ACTION LASTRA_WA_INIT:
Mission^.PPlace	:= cwa; (* valorizzo il punto di deposito *)
(* Aggiorno la struttura delle Lastre in missione *)
Mission^.Slab := WorkAreaState^[Mission^.PPick].Slab[WorkAreaState^[cwa].P];

NLastraDaPrelevare := WorkAreaState^[Mission^.PPick].P-1;
IF NLastraDaPrelevare >= 1 THEN
	NLastraDaPrelevare := 1 ;// añadido para probar
ELSE
	Errore.Code := ErrWA_NumPezzInPrelErrato;
	RETURN;
END_IF


				
Mission^.TPick 	:= TPICK_LASTRA;	// Assegno il tipo di Prelievo
Mission^.XDim 	:= Forming^[WorkAreaState^[Mission^.PPlace].F].PElement[NLastraDaPrelevare].XDim;// WorkAreaState^[Mission^.PPick].Slab[NLastraDaPrelevare].XDim;	// Assegno la dimensione X del pacco presente nel punto di prelievo designato
Mission^.YDim 	:= Forming^[WorkAreaState^[Mission^.PPlace].F].PElement[NLastraDaPrelevare].YDim;//WorkAreaState^[Mission^.PPick].Slab[NLastraDaPrelevare].YDim;	// Assegno la dimensione Y del pacco presente nel punto di prelievo designato
Mission^.ZDim 	:= Forming^[WorkAreaState^[Mission^.PPlace].F].PElement[NLastraDaPrelevare].ZDim;//WorkAreaState^[Mission^.PPick].Slab[NLastraDaPrelevare].ZDim; 	// Assegno la dimensione Z del pacco presente nel punto di prelievo designato
ppick := Mission^.PPick;

IF Mission^.XDim <=0	OR Mission^.YDim <= 0 THEN
	Errore.Code := ErrEsMisionSinDimesionPieza;
	RETURN;
END_IF
(* Valorizzazione del lato di prelievo nel caso di prelievo su cavallina *)
IF WorkareaState^[Mission^.PPick].Supporto.Tipologia = e_Tipo_Pallet.BUNDLE THEN //Se ho in prelievo il supporto di tipo bundle
	IF ppickOld <> Mission^.PPick THEN 	//Ad ogni cambio di postazione setto il valore del lato iniziale a 0
		TFClearApprendimento(ADR(WorkAreaState^[Mission^.PPick].Apprendimento));//Pulisco la struttura dell'apprendimento
		LatoPrelievo := 180;				//Vado a prelevare sul lato 180	
		TFWAM_CreaMissione_PrelLastraDaWA.Quota_FormaturaJ := 180; //Assegno la quota di 0° per il prelievo, in questo modo la pinza parte a fare il tasteggio in questa posizione					
		IF LatoPrelievo = 0 THEN
		(* Apprendimento lungo X *)
			WorkAreaState^[Mission^.PPick].Apprendimento.X.Lato0.Stato		:= APPRENDIMENTO_DISABILITATO;
			WorkAreaState^[Mission^.PPick].Apprendimento.Y.Lato0.Stato		:= APPRENDIMENTO_DA_ESEGUIRE;
		ELSIF LatoPrelievo = 180 THEN
			WorkAreaState^[Mission^.PPick].Apprendimento.X.Lato180.Stato	:= APPRENDIMENTO_DISABILITATO;
			WorkAreaState^[Mission^.PPick].Apprendimento.Y.Lato180.Stato	:= APPRENDIMENTO_DA_ESEGUIRE;
		END_IF
	ELSE
		LatoPrelievo := 180;				//Vado a prelevare sul lato 180	
		TFWAM_CreaMissione_PrelLastraDaWA.Quota_FormaturaJ := 180; //Assegno la quota di 0° per il prelievo, in questo modo la pinza parte a fare il tasteggio in questa posizione					
		IF LatoPrelievo = 0 THEN
		(* Apprendimento lungo X *)
			WorkAreaState^[Mission^.PPick].Apprendimento.X.Lato0.Stato		:= APPRENDIMENTO_DISABILITATO;
			IF WorkAreaState^[Mission^.PPick].Apprendimento.Y.Lato0.Stato <> APPRENDIMENTO_ESEGUITO THEN
				WorkAreaState^[Mission^.PPick].Apprendimento.Y.Lato0.Stato		:= APPRENDIMENTO_DA_ESEGUIRE;
			END_IF
		ELSIF LatoPrelievo = 180 THEN
			WorkAreaState^[Mission^.PPick].Apprendimento.X.Lato180.Stato	:= APPRENDIMENTO_DISABILITATO;
			IF WorkAreaState^[Mission^.PPick].Apprendimento.Y.Lato180.Stato <> APPRENDIMENTO_ESEGUITO THEN
				WorkAreaState^[Mission^.PPick].Apprendimento.Y.Lato180.Stato	:= APPRENDIMENTO_DA_ESEGUIRE;
			END_IF
		END_IF
	END_IF
ELSIF WorkareaState^[Mission^.PPick].Supporto.Tipologia = e_Tipo_Pallet.CAVALLETTO THEN //Se ho in prelievo il supporto di tipo cavalletto
	
	AguloDeRecogida := FunLadoTrabajoCaballete(Piezas_LadoA := 
						HMI_NumeroPezziPresentiCavallete[Mission^.PPick].HMI_NumeroPezziPresentiPostazione_A_Cavaleto , 
								Piezas_Ladob := HMI_NumeroPezziPresentiCavallete[Mission^.PPick].HMI_NumeroPezziPresentiPostazione_B_Cavaleto ,
								Recoger := TRUE ,dejar := FALSE ,GestionLadoTrabajo := WorkareaState^[Mission^.PPick].Supporto.TipoTrabajoLado_Cavallete);
	LatoPrelievo := AguloDeRecogida ;
	IF FALSE THEN 
			IF FormaturaAFRAMERT[WorkAreaState^[Mission^.PPlace].F].PElement[WorkAreaState^[Mission^.PPick].P-1].J > 90 THEN
				LatoPrelievo := 180;
			
			ELSIF FormaturaAFRAMERT[WorkAreaState^[Mission^.PPlace].F].PElement[WorkAreaState^[Mission^.PPick].P-1].J  < 90 THEN
				LatoPrelievo := 0;
			END_IF	
	END_IF
	
	IF ppickOld <> Mission^.PPick THEN 	//Ad ogni cambio di postazione setto il valore del lato iniziale a 0
		TFClearApprendimento(ADR(WorkAreaState^[Mission^.PPick].Apprendimento));//Pulisco la struttura dell'apprendimento
		TFWAM_CreaMissione_PrelLastraDaWA.Quota_FormaturaJ := 180; //Assegno la quota di 0° per il prelievo, in questo modo la pinza parte a fare il tasteggio in questa posizione					
		WorkAreaState^[Mission^.PPick].Apprendimento.X.Lato0.Stato		:= APPRENDIMENTO_DISABILITATO;
		WorkAreaState^[Mission^.PPick].Apprendimento.Y.Lato0.Stato		:= APPRENDIMENTO_DA_ESEGUIRE;
		WorkAreaState^[Mission^.PPick].Apprendimento.X.Lato180.Stato	:= APPRENDIMENTO_DISABILITATO;
		WorkAreaState^[Mission^.PPick].Apprendimento.Y.Lato180.Stato	:= APPRENDIMENTO_DA_ESEGUIRE;
	ELSE
		TFWAM_CreaMissione_PrelLastraDaWA.Quota_FormaturaJ := 180; //Assegno la quota di 0° per il prelievo, in questo modo la pinza parte a fare il tasteggio in questa posizione					
		IF LatoPrelievo = 0 THEN
		(* Apprendimento lungo X *)
			WorkAreaState^[Mission^.PPick].Apprendimento.X.Lato0.Stato		:= APPRENDIMENTO_DISABILITATO;
			IF WorkAreaState^[Mission^.PPick].Apprendimento.Y.Lato0.Stato <> APPRENDIMENTO_ESEGUITO THEN
				WorkAreaState^[Mission^.PPick].Apprendimento.Y.Lato0.Stato		:= APPRENDIMENTO_DA_ESEGUIRE;
				//WorkAreaState^[Mission^.PPick].Apprendimento.Y.Lato0.QuotaStart	:= 1000;
			END_IF
		ELSIF LatoPrelievo = 180 THEN
			WorkAreaState^[Mission^.PPick].Apprendimento.X.Lato180.Stato	:= APPRENDIMENTO_DISABILITATO;
			IF WorkAreaState^[Mission^.PPick].Apprendimento.Y.Lato180.Stato <> APPRENDIMENTO_ESEGUITO THEN
				WorkAreaState^[Mission^.PPick].Apprendimento.Y.Lato180.Stato	:= APPRENDIMENTO_DA_ESEGUIRE;
				//WorkAreaState^[Mission^.PPick].Apprendimento.Y.Lato180.QuotaStart	:= 1000;
			END_IF
		END_IF
	END_IF
ELSIF WorkareaState^[Mission^.PPick].Supporto.Tipologia <> e_Tipo_Pallet.CAVALLETTO AND WorkareaState^[Mission^.PPick].Supporto.Tipologia <> e_Tipo_Pallet.BUNDLE THEN //Se NON ho in prelievo il supporto di tipo cavalletto
	LatoPrelievo := 90; //Setto il lato di prelievo = 90
	IF ppickOld <> ppick THEN 	//Ad ogni cambio di postazione setto il valore del lato iniziale a 0
		TFClearApprendimento(ADR(WorkAreaState^[Mission^.PPick].Apprendimento));//Pulisco la struttura dell'apprendimento
	END_IF
	TFWAM_CreaMissione_PrelLastraDaWA.Quota_FormaturaJ := 90;//Assegno la quota di 90° per il prelievo, in questo modo la pinza preleverà in orizzontale
	IF WorkAreaState^[Mission^.PPick].Apprendimento.Z.Lato90.Stato <> APPRENDIMENTO_ESEGUITO THEN
		WorkAreaState^[Mission^.PPick].Apprendimento.Z.Lato90.Stato := APPRENDIMENTO_DA_ESEGUIRE;
		IF WorkareaState^[Mission^.PPick].Supporto.Tipologia = e_Tipo_Pallet.CASSA_STANDARD THEN 
			WorkAreaState^[Mission^.PPick].Apprendimento.Z.Lato90.QuotaStart 	:= 700;
		ELSE
			WorkAreaState^[Mission^.PPick].Apprendimento.Z.Lato90.QuotaStart 	:= 700;
		END_IF
	END_IF
END_IF

//Disabilito apprendimento in deposito se disabilitato
IF NOT HMI_AbilitaDepositoPaccoOrrizzontaleConTasteggio AND FALSE THEN
	WorkAreaState^[Mission^.PPick].Apprendimento.Z.Lato90.Stato := APPRENDIMENTO_DISABILITATO;	
END_IF

(* Memorizzo l'ultima postazione in cui è stato effettuato il prelievo *)
UltimaPostazioneInPrelievo := Mission^.PPick;
ppickOld := Mission^.PPick;

//Z prelievo a seconda della tipologia 
IF WorkareaState^[Mission^.PPick].Supporto.Tipologia = e_Tipo_Pallet.BUNDLE THEN //SE PRELIEVO SU BUNDLE O CASSA
	IF LatoPrelievo = 180 THEN
		AngoloPrelievo 					:= 180-2;
		AltezzaCentroLastraInclinata 	:=  	ABS((Mission^.YDim/2) * COS(DEG_TO_RAD(AngoloPrelievo)));
		QuotaLastraYRealTimePrelievo 			:= FormaturaBundleRT[WorkAreaProductionList^[Mission^.PPlace].NumeroListaAssociata].PElement[WorkAreaState^[Mission^.PPick].P-1].Y;
		QuotaLastraZRealTimePrelievo 			:= FormaturaBundleRT[WorkAreaProductionList^[Mission^.PPlace].NumeroListaAssociata].PElement[WorkAreaState^[Mission^.PPick].P-1].Z (*+  (*Dimensioni_Pinza.DimTraveVerticale / 2*) CuotaOffSetZRecogidaBundel *);
	ELSIF LatoPrelievo = 0 THEN
		AngoloPrelievo 							:= 2;
		AltezzaCentroLastraInclinata 			:=  ABS((Mission^.YDim/2) * COS(DEG_TO_RAD(AngoloPrelievo)));
		IF TRUE THEN 
			QuotaLastraYRealTimePrelievo 			:= FormaturaBundleRT[WorkAreaProductionList^[Mission^.PPlace].NumeroListaAssociata].PElement[WorkAreaState^[Mission^.PPick].P_Cava.HMI_NumeroPezziPresentiPostazione_A_Cavaleto-1].CooCavallete.LadoA.CoordenadaFinale_Y;
			QuotaLastraZRealTimePrelievo 			:= FormaturaBundleRT[WorkAreaProductionList^[Mission^.PPlace].NumeroListaAssociata].PElement[WorkAreaState^[Mission^.PPick].P_Cava.HMI_NumeroPezziPresentiPostazione_A_Cavaleto-1].CooCavallete.LadoA.CoordenadaFinale_Z;(*+  (*Dimensioni_Pinza.DimTraveVerticale / 2*) CuotaOffSetZRecogidaBundel *);
		ELSE
			QuotaLastraYRealTimePrelievo 			:= FormaturaBundleRT[WorkAreaProductionList^[Mission^.PPlace].NumeroListaAssociata].PElement[WorkAreaState^[Mission^.PPick].P-1].Y;
			QuotaLastraZRealTimePrelievo 			:= FormaturaBundleRT[WorkAreaProductionList^[Mission^.PPlace].NumeroListaAssociata].PElement[WorkAreaState^[Mission^.PPick].P-1].Z (*+ (*Dimensioni_Pinza.DimTraveVerticale / 2*) CuotaOffSetZRecogidaBundel*) ;		
			
		END_IF
		
	ELSE
		AngoloPrelievo := 90;
		AltezzaCentroLastraInclinata := 0;
		QuotaLastraZRealTimePrelievo := 0;
		QuotaLastraYRealTimePrelievo := 0;
	END_IF
ELSIF WorkareaState^[Mission^.PPick].Supporto.Tipologia = e_Tipo_Pallet.CAVALLETTO THEN
	IF LatoPrelievo = 180 THEN
		AngoloPrelievo 					:= 180-2;
		AltezzaCentroLastraInclinata 	:= ABS((Mission^.YDim/2) * COS(DEG_TO_RAD(AngoloPrelievo)));
		IF TRUE THEN
			QuotaLastraYRealTimePrelievo 			:= FormaturaAFRAMERT[WorkAreaProductionList^[Mission^.PPlace].NumeroListaAssociata].PElement[WorkAreaState^[Mission^.PPick].P_Cava.HMI_NumeroPezziPresentiPostazione_B_Cavaleto-1].CooCavallete.LadoB.CoordenadaFinale_Y;
			QuotaLastraZRealTimePrelievo 			:= FormaturaAFRAMERT[WorkAreaProductionList^[Mission^.PPlace].NumeroListaAssociata].PElement[WorkAreaState^[Mission^.PPick].P_Cava.HMI_NumeroPezziPresentiPostazione_B_Cavaleto-1].CooCavallete.LadoB.CoordenadaFinale_Z;(*+  (*Dimensioni_Pinza.DimTraveVerticale / 2*) CuotaOffSetZRecogidaBundel *);
		ELSE
 			QuotaLastraYRealTimePrelievo 			:= FormaturaAFRAMERT[WorkAreaProductionList^[Mission^.PPlace].NumeroListaAssociata].PElement[WorkAreaState^[Mission^.PPick].P-1].Y;
			QuotaLastraZRealTimePrelievo 			:= FormaturaAFRAMERT[WorkAreaProductionList^[Mission^.PPlace].NumeroListaAssociata].PElement[WorkAreaState^[Mission^.PPick].P-1].Z + (*Dimensioni_Pinza.DimTraveVerticale / 2*) CuotaOffSetZRecogidaCaballete;
		END_IF
	ELSIF LatoPrelievo = 0 THEN
		AngoloPrelievo 					:= 3;
		AltezzaCentroLastraInclinata 	:= ABS((Mission^.YDim/2) * COS(DEG_TO_RAD(AngoloPrelievo)));
		IF TRUE THEN 
			QuotaLastraYRealTimePrelievo 			:= FormaturaAFRAMERT[WorkAreaProductionList^[Mission^.PPlace].NumeroListaAssociata].PElement[WorkAreaState^[Mission^.PPick].P_Cava.HMI_NumeroPezziPresentiPostazione_A_Cavaleto-1].CooCavallete.LadoA.CoordenadaFinale_Y;
			QuotaLastraZRealTimePrelievo 			:= FormaturaAFRAMERT[WorkAreaProductionList^[Mission^.PPlace].NumeroListaAssociata].PElement[WorkAreaState^[Mission^.PPick].P_Cava.HMI_NumeroPezziPresentiPostazione_A_Cavaleto-1].CooCavallete.LadoA.CoordenadaFinale_Z;(*+  (*Dimensioni_Pinza.DimTraveVerticale / 2*) CuotaOffSetZRecogidaBundel *);
		ELSE
			QuotaLastraYRealTimePrelievo 			:= FormaturaAFRAMERT[WorkAreaProductionList^[Mission^.PPlace].NumeroListaAssociata].PElement[WorkAreaState^[Mission^.PPick].P-1].Y;
			QuotaLastraZRealTimePrelievo 			:= FormaturaAFRAMERT[WorkAreaProductionList^[Mission^.PPlace].NumeroListaAssociata].PElement[WorkAreaState^[Mission^.PPick].P-1].Z (*+ (*Dimensioni_Pinza.DimTraveVerticale / 2*) CuotaOffSetZRecogidaCaballete *);
		END_IF
	ELSE
		AngoloPrelievo := 90;
		AltezzaCentroLastraInclinata := 0;
		QuotaLastraZRealTimePrelievo := 0;
		QuotaLastraYRealTimePrelievo := 0;
	END_IF
ELSE
	IF LatoPrelievo = 90 THEN		
		AngoloPrelievo := 90;
		AltezzaCentroLastraInclinata := 0;
		QuotaLastraZRealTimePrelievo := 0;
		QuotaLastraYRealTimePrelievo := 0;
	ELSE
		Errore.Code := ErrWA_SupportoInPrelivoNonPrevisto;
	END_IF
END_IF

//CALCOLO INGOMBRI PINZA						

;
//OffSetZRecogidaEnAngulo				:=  -20 ;					
//ScostamentoVerticalePuntoCentrale := ABS(Dimensioni_Pinza.Spessore * COS(deg_to_rad(-90+AngoloPrelievo))-Dimensioni_Pinza.Spessore);

// Calculo Del Ingombro Pinza Mision Recogida lastra
TFCalcoliIngombroPinza(Mission := Mission,
						WorkAreaManager := WorkAreaManager,
						WorkAreaState := ADR(WorkAreaState),
						ModuleAX_J := ModuleAX_J,
						AngoloRotazioneDestinazionePinza:= LatoPrelievo,//Forming^[WorkAreaState^[Mission^.PPlace].F].PElement[WorkAreaState^[Mission^.PPlace].P].J+2,
						IngombroX_Pos 				:= ADR(IngombroX_Pos),
						IngombroY_Pos 				:= ADR(IngombroY_Pos),
						IngombroX_Neg 				:= ADR(IngombroX_Neg),
						IngombroY_Neg 				:= ADR(IngombroY_Neg),
						IngombroZ_Pos 				:= ADR(IngombroZ_Pos),
						IngombroZ_Neg 				:= ADR(IngombroZ_Neg),
						IngombroY_Tot 				:= ADR(IngombroY_Tot),
						IngombroDestinazioneX_Pos 	:= ADR(IngombroDestinazioneX_Pos),
						IngombroDestinazioneY_Pos 	:= ADR(IngombroDestinazioneY_Pos),
						IngombroDestinazioneX_Neg 	:= ADR(IngombroDestinazioneX_Neg),
						IngombroDestinazioneY_Neg 	:= ADR(IngombroDestinazioneY_Neg),
						IngombroDestinazioneZ_Pos 	:= ADR(IngombroDestinazioneZ_Pos),
						IngombroDestinazioneZ_Neg 	:= ADR(IngombroDestinazioneZ_Neg),
						IngombroMaxX_Pos 			:= ADR(IngombroMaxX_Pos),
						IngombroMaxY_Pos 			:= ADR(IngombroMaxY_Pos),
						IngombroMaxX_Neg 			:= ADR(IngombroMaxX_Neg),
						IngombroMaxY_Neg 			:= ADR(IngombroMaxY_Neg),
						IngombroMaxZ_Pos 			:= ADR(IngombroMaxZ_Pos),
						IngombroMaxZ_Neg 			:= ADR(IngombroMaxZ_Neg),
						IngombroY_Pos_0  			:= ADR(IngombroY_Pos_0),		 		
						IngombroY_Neg_180 			:= ADR(IngombroY_Neg_180),
						IngombroY_Neg_0 			:= ADR(IngombroY_Neg_0),	
						IngombroY_Pos_180 			:= ADR(IngombroY_Pos_180),
						ScostamentoVerticalePuntoCentrale := ADR(ScostamentoVerticalePuntoCentrale));





(* Assegnazione quote alla Missione *)
TFWAM_CreaMissione_PrelLastraDaWA(NPosInLavoro				:= Mission^.PPick, //Numero Postazione di lavoro
									Angolo_Destinazione 	:= LatoPrelievo, //Angolo di deposito dell'elemento
									PosizioneAttuale_X      := ModuleAX_X^.Ax^.Status.ActPosition, //Posizione attuale asse X
									TipologiaTraiettoria    := TRAIETTORIA_CON_APPROCCIO,//Forming^[WorkAreaState^[cwa].F].PElement[WorkAreaState^[cwa].P].Trajectory,
									Apprendimento			:= WorkAreaState^[Mission^.PPick].Apprendimento,
									CicloDiPrelievo         := TRUE,
									HmaxElemento			:= WorkAreaState^[Mission^.PPick].Supporto.HMAX,
									Offset_Apprendimento_X 	:= 0,//OffsetApprendimento.Lastra.X, //Offset X Postazione,
									Offset_Apprendimento_Y 	:= OffsetApprendimento.Lastra.Y, //Offset Y Postazione
									Offset_Apprendimento_Z 	:= OffsetApprendimento.Lastra.Z, //Offset Z Postazione
									Offset_Apprendimento_J 	:= 0,//OffsetApprendimento.Lastra.J, //Offset J Postazione

									Quota_PostX				:= WorkArea^[Mission^.PPick].X, //Quota X Postazione
									Quota_PostY				:= WorkArea^[Mission^.PPick].Y, //Quota Y Postazione
									Quota_PostZ				:= WorkArea^[Mission^.PPick].Z, //Quota Z Postazione
									Quota_PostJ				:= WorkArea^[Mission^.PPick].Rx, //Quota J Postazione
									
									Offset_Postazione_X 	:= WorkAreaOffset^[Mission^.PPick].X, //Offset X Postazione
									Offset_Postazione_Y 	:= WorkAreaOffset^[Mission^.PPick].Y, //Offset Y Postazione
									Offset_Postazione_Z 	:= WorkAreaOffset^[Mission^.PPick].Z, //Offset Z Postazione
									Offset_Postazione_J 	:= WorkAreaOffset^[Mission^.PPick].Rx, //Offset J Postazione
									
									Pallet_DimX				:= WorkAreaState^[Mission^.PPick].Supporto.XDim, //Dimensione X Pallet
									Pallet_DimY				:= WorkAreaState^[Mission^.PPick].Supporto.YDim, //Dimensione Y Pallet
									Pallet_DimZ				:= WorkAreaState^[Mission^.PPick].Supporto.ZDim, //Dimensione Z Pallet
									Pallet_DimBaseUtile		:= WorkAreaState^[Mission^.PPick].Supporto.DimBaseUtile, //Dimensione Z Pallet
									
									Offset_Pallet_X_0		:= 0,//Forming^[WorkAreaState^[Mission^.PPlace].F].Pallet.OFSDE_X0, //Offset X Pallet o Casse
									Offset_Pallet_Y_0		:= 0,//Forming^[WorkAreaState^[Mission^.PPlace].F].Pallet.OFSDE_Y0, //Offset Y Pallet o Casse 
									Offset_Pallet_Z_0		:= OffSetZRecogidaEnAngulo0,//Forming^[WorkAreaState^[Mission^.PPlace].F].Pallet.OFSDE_Z0, //Offset Z Pallet o Casse + è grande + il deposito si distanzia dal supporto
									Offset_Pallet_J_0		:= 0,//Forming^[WorkAreaState^[Mission^.PPlace].F].Pallet.OFSDE_J0, //Offset J Pallet o Casse + è grande + la lastra sarà inclinata verso l'angolo crescente
															   
									Offset_Pallet_X_90		:= 0,//Forming^[WorkAreaState^[Mission^.PPlace].F].Pallet.OFSDE_X90, //Offset X Pallet lato 0-90 
									Offset_Pallet_Y_90		:= 0,//Forming^[WorkAreaState^[Mission^.PPlace].F].Pallet.OFSDE_Y90, //Offset Y Pallet lato 0-90 + è grande + il deposito si distanzia dal supporto
									Offset_Pallet_Z_90		:= 0,//Forming^[WorkAreaState^[Mission^.PPlace].F].Pallet.OFSDE_Z90, //Offset Z Pallet lato 0-90 + è grande + il deposito si distanzia dal supporto
									Offset_Pallet_J_90		:= 0,//Forming^[WorkAreaState^[Mission^.PPlace].F].Pallet.OFSDE_J90, //Offset J Pallet lato 0-90 + è grande + la lastra sarà inclinata in fase di deposito
															  
									Offset_Pallet_X_180		:= 0,//Forming^[WorkAreaState^[Mission^.PPlace].F].Pallet.OFSDE_X180, //Offset X Pallet lato 90-180
									Offset_Pallet_Y_180		:= 0,//Forming^[WorkAreaState^[Mission^.PPlace].F].Pallet.OFSDE_Y180, //Offset Y Pallet lato 90-180 + è grande + il deposito si distanzia dal supporto
									Offset_Pallet_Z_180		:= OffSetZRecogidaEnAngulo180,//Forming^[WorkAreaState^[Mission^.PPlace].F].Pallet.OFSDE_Z180, //Offset Z Pallet lato 90-180 + è grande + il deposito si distanzia dal supporto
									Offset_Pallet_J_180		:= 0,//Forming^[WorkAreaState^[Mission^.PPlace].F].Pallet.OFSDE_J180, //Offset J Pallet lato 90-180 + è grande + la lastra sarà inclinata in fase di deposito
									
									Quota_FormaturaX 		:= 0,//Quota  X da Formatura
									Quota_FormaturaY 		:= ABS(QuotaLastraYRealTimePrelievo),//Quota  Y da Formatura
									Quota_FormaturaZ 		:= QuotaLastraZRealTimePrelievo,//Quota  Z da Formatura
									Quota_FormaturaJ 		:= LatoPrelievo,//Quota  Z da Formatura
									
									Distanza_ApproccioFormaturaX 		:= PickPlaceParameters^.XPickApproach,
									Distanza_ApproccioFormaturaY 		:= PickPlaceParameters^.YPickApproach, 
									Distanza_ApproccioFormaturaZ 		:= PickPlaceParameters^.ZPickApproach,
									Distanza_ApproccioFormaturaJ 		:= PickPlaceParameters^.JPickApproach,
									
									Quota_DestX 			=> Mission^.XPick, //Quota DESTINAZIONE X
									Quota_DestY 			=> Mission^.YPick, //Quota DESTINAZIONE Y
									Quota_DestZ 			=> Mission^.ZPick, //Quota DESTINAZIONE Z
									Quota_DestJ 			=> Mission^.JPick, //Quota DESTINAZIONE J	
									
									Quota_ApproccioDestX 	=> Mission^.XPickApproach, //Quota APPROCCIO di DESTINAZIONE X
									Quota_ApproccioDestY 	=> Mission^.YPickApproach, //Quota APPROCCIO di DESTINAZIONE Y
									Quota_ApproccioDestZ 	=> Mission^.ZPickApproach, //Quota APPROCCIO di DESTINAZIONE Z
									Quota_ApproccioDestJ 	=> Mission^.JPickApproach);//Quota APPROCCIO di DESTINAZIONE J	

//Valorizziamo il preleivo di z a una quota positiva per evitare errori di interferenza									
IF LatoPrelievo = 90 THEN
	IF Mission^.ZPick <= 0 THEN
		Mission^.ZPick := ModuleAX_Z^.AxisPar^.MinPosition;
	END_IF
END_IF 		
//
IF LatoPrelievo = 180 THEN
	
	IF HMI_OffsetDepositoLastra.J180 = 0 OR  HMI_OffsetDepositoLastra.J180 < 0 THEN 
		Mission^.JPick := 180 - 2;
	ELSIF HMI_OffsetDepositoLastra.J180 <= 4 AND   HMI_OffsetDepositoLastra.J180 > 0 THEN 
		Mission^.JPick := 180 - HMI_OffsetDepositoLastra.J180;
	ELSE 
		Mission^.JPick := 180 - 2;	
	END_IF
	


	
	
	
	//IF WorkAreaState^[Mission^.PPick].Apprendimento.Y.Lato180.Stato = APPRENDIMENTO_ESEGUITO THEN
	//	Mission^.YPickApproach	:= MIN(Mission^.YPickApproach,WorkAreaState^[Mission^.PPick].Supporto.YDim + IngombroDestinazioneY_Neg);
	//ELSE
	//	Mission^.YPickApproach	:= WorkArea^[Mission^.PPick].Y + WorkAreaState^[Mission^.PPick].Supporto.YDim + IngombroDestinazioneY_Neg - 50;
	//end_if
	//&&&&&&&&&&&&&&&&&&&&&&&&&&&&&&&&&&&&&&&&&&&&&&&&&&&&&&&&&&&&&&&&&&&&&&&&&&&&&
	//Mission^.YPick 				:= Mission^.YPick - 80 ;	// modificado = 200
	//&&&&&&&&&&&&&&&&&&&&&&&&&&&&&&&&&&&&&&&&&&&&&&&&&&&&&&&&&&&&&&&&&&&&&&&&&&&&&&&&&&&&
	IF WorkareaState^[Mission^.PPick].Supporto.Tipologia = e_Tipo_Pallet.BUNDLE THEN //SE PRELIEVO SU BUNDLE O CASSA
		Y_PuntoPrelievo180 := Mission^.YPick ;
			Z_PuntoPrelievo180Bundle    := Mission^.ZPick ;
		 IF Mission^.YDim  < 1300 THEN
			Mission^.YPick 				:= Mission^.YPick - (80  ) ; //(Dimensioni_Pinza.DimTraveVerticale /2) (*-80*);	// modificado = 200
			Mission^.ZPick				:= Mission^.ZPick + (15 +25) ;
			Mission^.ZPickApproach		:= Mission^.ZPick;
			ELSE
				
			Mission^.YPick 				:= Mission^.YPick  - (45) ; //(Dimensioni_Pinza.DimTraveVerticale /2) (*-80*);	// modificado = 200
 			Mission^.ZPick				:= Mission^.ZPick + 15 ;
			Mission^.ZPickApproach		:= Mission^.ZPick;
		 END_IF
		
	
		
	ELSIF WorkareaState^[Mission^.PPick].Supporto.Tipologia = e_Tipo_Pallet.CAVALLETTO THEN //Se ho in prelievo il supporto di tipo cavalletto	
		Y_PuntoPrelievo180 := Mission^.YPick ;
		Z_PuntoPrelievo180Bundle    := Mission^.ZPick ;
		IF Mission^.YDim  < 1300 THEN
				Mission^.YPick 				:= Mission^.YPick - (Dimensioni_Pinza.DimTraveVerticale -35) ;//(Dimensioni_Pinza.DimTraveVerticale /2) (*-70*)  ;	// modificado = 200
				Mission^.ZPick				:= Mission^.ZPick + (25 +20) ;
				Mission^.ZPickApproach		:= Mission^.ZPick;		
			ELSE
				Mission^.YPick 				:= Mission^.YPick - 60 ; //(Dimensioni_Pinza.DimTraveVerticale /2) (*-70*)  ;	// modificado = 200
				Mission^.ZPick				:= Mission^.ZPick + 28 ;
				Mission^.ZPickApproach		:= Mission^.ZPick;		
			
		END_IF
		
		
	END_IF

ELSIF LatoPrelievo = 0 THEN
	//Mission^.JPick := 3;
	IF HMI_OffsetDepositoLastra.J0 > 4 THEN 
		Mission^.JPick := 4;
	ELSIF HMI_OffsetDepositoLastra.J0 <> 0 THEN 
		Mission^.JPick := HMI_OffsetDepositoLastra.J0;	
	ELSIF HMI_OffsetDepositoLastra.J0 = 0 THEN 
		Mission^.JPick := 3;	
	END_IF
	Y_PuntoPrelievo0 := Mission^.YPick ;
	
	Z_PuntoPrelievo180Bundle    := Mission^.ZPick ;
	IF Mission^.YDim  < 1300 THEN
			Mission^.YPick 				:= Mission^.YPick -0 ; // + 50 (*+ 50 *);
			Mission^.ZPick				:= Mission^.ZPick + (20) ; // pieza pequeña
			Mission^.ZPickApproach		:= Mission^.ZPick;
		ELSE
			Mission^.YPick 				:= Mission^.YPick  + 25; // + 50 (*+ 50 *);
			Mission^.ZPick				:= Mission^.ZPick + 12 ;
			Mission^.ZPickApproach		:= Mission^.ZPick;	
	END_IF
	
	
	
END_IF											 			
//									
IF TFWAM_CreaMissione_PrelLastraDaWA.Errore.Code > 0 THEN
	Errore := TFWAM_CreaMissione_PrelLastraDaWA.Errore;
	WorkAreaManager^.State 	:= WAMANAGER_NOP;	// setto lo stato del WAMANAGER
	RETURN;//EXIT;
END_IF	

(* Valorizzazione del lato di prelievo nel caso di depostio su cavallina *)
IF WorkareaState^[Mission^.PPlace].Supporto.Tipologia = e_Tipo_Pallet.CAVALLETTO THEN //Se ho in prelievo il supporto di tipo cavalletto
	
	AguloDeDeposito := FunLadoTrabajoCaballete(Piezas_LadoA := 
						HMI_NumeroPezziPresentiCavallete[Mission^.PPlace].HMI_NumeroPezziPresentiPostazione_A_Cavaleto , 
								Piezas_Ladob := HMI_NumeroPezziPresentiCavallete[Mission^.PPlace].HMI_NumeroPezziPresentiPostazione_B_Cavaleto ,
								Recoger := FALSE ,dejar := TRUE, GestionLadoTrabajo := WorkareaState^[Mission^.PPlace].Supporto.TipoTrabajoLado_Cavallete);
	LatoDeposito := AguloDeDeposito ;

	IF FALSE THEN
		IF FormaturaAFRAMERT[WorkAreaState^[Mission^.PPlace].F].PElement[WorkAreaState^[Mission^.PPlace].P].J > 90 THEN
			LatoDeposito := 180;
		
		ELSIF FormaturaAFRAMERT[WorkAreaState^[Mission^.PPlace].F].PElement[WorkAreaState^[Mission^.PPlace].P].J  < 90 THEN
			LatoDeposito := 0;
		END_IF
	END_IF
	
	
ELSIF WorkareaState^[Mission^.PPlace].Supporto.Tipologia = e_Tipo_Pallet.BUNDLE THEN
	LatoDeposito := 180;
ELSIF WorkareaState^[Mission^.PPlace].Supporto.Tipologia <> e_Tipo_Pallet.CAVALLETTO AND WorkareaState^[Mission^.PPlace].Supporto.Tipologia <> e_Tipo_Pallet.BUNDLE THEN //Se NON ho in prelievo il supporto di tipo cavalletto
	IF PplaceOld <> Mission^.PPlace THEN 	//Ad ogni cambio di postazione setto il valore del lato iniziale a 0
		TFClearApprendimento(ADR(WorkAreaState^[Mission^.PPlace].Apprendimento));//Pulisco la struttura dell'apprendimento
	END_IF
	LatoDeposito := 90; //Setto il lato di prelievo = 90
	TFWAM_CreaMissione_PrelLastraDaWA.Quota_FormaturaJ := 90;//Assegno la quota di 90° per il prelievo, in questo modo la pinza preleverà in orizzontale
	IF WorkAreaState^[Mission^.PPlace].Apprendimento.Z.Lato90.Stato <> APPRENDIMENTO_ESEGUITO THEN
		WorkAreaState^[Mission^.PPlace].Apprendimento.Z.Lato90.Stato := APPRENDIMENTO_DA_ESEGUIRE;
		IF WorkareaState^[Mission^.PPlace].Supporto.Tipologia = e_Tipo_Pallet.CASSA_STANDARD THEN 
			WorkAreaState^[Mission^.PPlace].Apprendimento.Z.Lato90.QuotaStart 	:= 700;
		ELSE
			WorkAreaState^[Mission^.PPlace].Apprendimento.Z.Lato90.QuotaStart 	:= 700;
		END_IF
	END_IF
END_IF

//Disabilito apprendimento in deposito se disabilitato
IF NOT HMI_AbilitaDepositoPaccoOrrizzontaleConTasteggio AND FALSE THEN
	WorkAreaState^[Mission^.PPlace].Apprendimento.Z.Lato90.Stato := APPRENDIMENTO_DISABILITATO;	
END_IF

//mettiamo un offset sul deposito bundle
IF LatoDeposito = 180 THEN
	TFWAM_CreaMissione_DepLastraDaWA.Offset_Pallet_Y_0 := 0;// HMI_OffsetDepositoLastra.Y0;
	TFWAM_CreaMissione_DepLastraDaWA.Offset_Pallet_Z_0 := 0;//HMI_OffsetDepositoLastra.Z0;
	TFWAM_CreaMissione_DepLastraDaWA.Offset_Pallet_Y_0 := 0;

	TFWAM_CreaMissione_DepLastraDaWA.Offset_Pallet_Y_180 := HMI_OffsetDepositoLastra.Y180;
	TFWAM_CreaMissione_DepLastraDaWA.Offset_Pallet_Z_180 := HMI_OffsetDepositoLastra.Z180;
	TFWAM_CreaMissione_DepLastraDaWA.Offset_Pallet_Z_90  := 0;
	AngoloDepositoLastra := 180; // := 180-1; Modificado 16-6-2025
ELSIF LatoDeposito = 90 THEN
	TFWAM_CreaMissione_DepLastraDaWA.Offset_Pallet_Y_180 := 0;
	TFWAM_CreaMissione_DepLastraDaWA.Offset_Pallet_Z_180 := 0;
	TFWAM_CreaMissione_DepLastraDaWA.Offset_Pallet_Y_180 := 0;
	IF NOT HMI_AbilitaDepositoPaccoOrrizzontaleConTasteggio THEN
		TFWAM_CreaMissione_DepLastraDaWA.Offset_Pallet_Z_90  := (* 30 +*) HMI_OffsetDepositoLastra.Z90; // quitado el ´30
	ELSE
		TFWAM_CreaMissione_DepLastraDaWA.Offset_Pallet_Z_90  := 0;
	END_IF
	AngoloDepositoLastra := 90;
ELSIF LatoDeposito = 0 THEN
	TFWAM_CreaMissione_DepLastraDaWA.Offset_Pallet_Y_180 := 0;
	TFWAM_CreaMissione_DepLastraDaWA.Offset_Pallet_Z_180 := 0;
	TFWAM_CreaMissione_DepLastraDaWA.Offset_Pallet_Y_180 := 0;

	//POMGO EL MISMO OFFSET EN Z PARA CAVALINA TANTO EN 0 COMO 180 
	//@@@@@@@@@@@@@@@@@@@@@@Para Quitar@@@@@@@@@@@@@@@@@@@@@@@@@@@@@@@@@@@@@@@@@@@@@@@
	//HMI_OffsetDepositoLastra.Z0 :=HMI_OffsetDepositoLastra.Z180 +10 ;
	//@@@@@@@@@@@@@@@@@@@@@@@@@@@@@@@@@@@@@@@@@@@@@@@@@@@@@@@@@@@@@@@@@@@@@
	TFWAM_CreaMissione_DepLastraDaWA.Offset_Pallet_Y_0 := HMI_OffsetDepositoLastra.Y0;
	TFWAM_CreaMissione_DepLastraDaWA.Offset_Pallet_Z_0 := HMI_OffsetDepositoLastra.Z0;
	TFWAM_CreaMissione_DepLastraDaWA.Offset_Pallet_Z_90  := 0;
	AngoloDepositoLastra := 1;
END_IF
// Calculo Del Ingombro Pinza Mision deposito lastra
TFCalcoliIngombroPinza(Mission := Mission,
						WorkAreaManager := WorkAreaManager,
						WorkAreaState := ADR(WorkAreaState),
						ModuleAX_J := ModuleAX_J,
						AngoloRotazioneDestinazionePinza:= AngoloDepositoLastra,//Forming^[WorkAreaState^[Mission^.PPlace].F].PElement[WorkAreaState^[Mission^.PPlace].P].J+2,
						IngombroX_Pos 				:= ADR(IngombroX_Pos),
						IngombroY_Pos 				:= ADR(IngombroY_Pos),
						IngombroX_Neg 				:= ADR(IngombroX_Neg),
						IngombroY_Neg 				:= ADR(IngombroY_Neg),
						IngombroZ_Pos 				:= ADR(IngombroZ_Pos),
						IngombroZ_Neg 				:= ADR(IngombroZ_Neg),
						IngombroY_Tot 				:= ADR(IngombroY_Tot),
						IngombroDestinazioneX_Pos 	:= ADR(IngombroDestinazioneX_Pos),
						IngombroDestinazioneY_Pos 	:= ADR(IngombroDestinazioneY_Pos),
						IngombroDestinazioneX_Neg 	:= ADR(IngombroDestinazioneX_Neg),
						IngombroDestinazioneY_Neg 	:= ADR(IngombroDestinazioneY_Neg),
						IngombroDestinazioneZ_Pos 	:= ADR(IngombroDestinazioneZ_Pos),
						IngombroDestinazioneZ_Neg 	:= ADR(IngombroDestinazioneZ_Neg),
						IngombroMaxX_Pos 			:= ADR(IngombroMaxX_Pos),
						IngombroMaxY_Pos 			:= ADR(IngombroMaxY_Pos),
						IngombroMaxX_Neg 			:= ADR(IngombroMaxX_Neg),
						IngombroMaxY_Neg 			:= ADR(IngombroMaxY_Neg),
						IngombroMaxZ_Pos 			:= ADR(IngombroMaxZ_Pos),
						IngombroMaxZ_Neg 			:= ADR(IngombroMaxZ_Neg),
						IngombroY_Pos_0  			:= ADR(IngombroY_Pos_0),		 		
						IngombroY_Neg_180 			:= ADR(IngombroY_Neg_180),
						IngombroY_Neg_0 			:= ADR(IngombroY_Neg_0),	
						IngombroY_Pos_180 			:= ADR(IngombroY_Pos_180),
						ScostamentoVerticalePuntoCentrale := ADR(ScostamentoVerticalePuntoCentrale));

ScostamentoVerticalePuntoCentrale := ABS(Dimensioni_Pinza.Spessore * COS(deg_to_rad(-90+AngoloDepositoLastra))-Dimensioni_Pinza.Spessore);		

//Z prelievo a seconda della tipologia 
IF WorkareaState^[Mission^.PPlace].Supporto.Tipologia = e_Tipo_Pallet.BUNDLE THEN //Se ho in DEPOSITO il supporto di tipo BUNDLE
	IF LatoDeposito <> 90 THEN
		QuotaLastraYRealTimeDeposito 		:= FormaturaBundleRT[WorkAreaProductionList^[Mission^.PPlace].NumeroListaAssociata].PElement[WorkAreaState^[Mission^.PPlace].P].Y;
		QuotaLastraZRealTimeDeposito 		:= FormaturaBundleRT[WorkAreaProductionList^[Mission^.PPlace].NumeroListaAssociata].PElement[WorkAreaState^[Mission^.PPlace].P].Z;
	ELSE
		Errore.Code := ErrWA_SupportoInPrelivoNonPrevisto;
	END_IF
ELSIF WorkareaState^[Mission^.PPlace].Supporto.Tipologia = e_Tipo_Pallet.CAVALLETTO THEN //Se ho in DEPOSITO il supporto di tipo CAVALLETTO
	IF LatoDeposito = 0 THEN 
		QuotaLastraYRealTimeDeposito 			:= FormaturaAFRAMERT[WorkAreaProductionList^[Mission^.PPlace].NumeroListaAssociata].PElement[WorkAreaState^[Mission^.PPlace].P_Cava.HMI_NumeroPezziPresentiPostazione_A_Cavaleto].CooCavallete.LadoA.CoordenadaFinale_Y;
		QuotaLastraZRealTimeDeposito			:= FormaturaAFRAMERT[WorkAreaProductionList^[Mission^.PPlace].NumeroListaAssociata].PElement[WorkAreaState^[Mission^.PPlace].P_Cava.HMI_NumeroPezziPresentiPostazione_A_Cavaleto].CooCavallete.LadoA.CoordenadaFinale_Z;
	ELSIF LatoDeposito = 180   THEN 
		QuotaLastraYRealTimeDeposito 			:= FormaturaAFRAMERT[WorkAreaProductionList^[Mission^.PPlace].NumeroListaAssociata].PElement[WorkAreaState^[Mission^.PPlace].P_Cava.HMI_NumeroPezziPresentiPostazione_B_Cavaleto].CooCavallete.LadoB.CoordenadaFinale_Y;
		QuotaLastraZRealTimeDeposito			:= FormaturaAFRAMERT[WorkAreaProductionList^[Mission^.PPlace].NumeroListaAssociata].PElement[WorkAreaState^[Mission^.PPlace].P_Cava.HMI_NumeroPezziPresentiPostazione_B_Cavaleto].CooCavallete.LadoB.CoordenadaFinale_Z;
	ELSE
		Errore.Code := ErrWA_SupportoInPrelivoNonPrevisto;	
	END_IF

	IF FALSE THEN 
		IF LatoDeposito <> 90 THEN
			QuotaLastraYRealTimeDeposito 		:= FormaturaAFRAMERT[WorkAreaProductionList^[Mission^.PPlace].NumeroListaAssociata].PElement[WorkAreaState^[Mission^.PPlace].P].Y;
			QuotaLastraZRealTimeDeposito 		:= FormaturaAFRAMERT[WorkAreaProductionList^[Mission^.PPlace].NumeroListaAssociata].PElement[WorkAreaState^[Mission^.PPlace].P].Z;
		ELSE
			Errore.Code := ErrWA_SupportoInPrelivoNonPrevisto;
		END_IF
	END_IF
	
	
	
ELSE
	QuotaLastraZRealTimeDeposito := Forming^[WorkAreaState^[Mission^.PPlace].F].PElement[WorkAreaState^[Mission^.PPlace].P].Z;
	QuotaLastraYRealTimeDeposito := ABS(Forming^[WorkAreaState^[Mission^.PPlace].F].PElement[WorkAreaState^[Mission^.PPlace].P].Y);
END_IF	

IF WorkAreaState^[Mission^.PPlace].Supporto.Tipologia = CAVALLETTO THEN
	OffSetY180Cavallete := 0 ;	
	ELSE 
	OffSetY180Cavallete := 0 ;	
	
END_IF


(* Valorizzazione quote di deposito Ciclo Lastra *)
TFWAM_CreaMissione_DepLastraDaWA(NPosInLavoro			:= Mission^.PPlace, //Numero Postazione di lavoro
								Angolo_Destinazione 	:= LatoDeposito, //Angolo di deposito dell'elemento
								PosizioneAttuale_X      := ModuleAX_X^.Ax^.Status.ActPosition, //Posizione attuale asse X
								TipologiaTraiettoria    := TRAIETTORIA_CON_APPROCCIO,//Forming^[WorkAreaState^[cwa].F].PElement[WorkAreaState^[cwa].P].Trajectory,
								Apprendimento			:= WorkAreaState^[Mission^.PPlace].Apprendimento,
								CicloDiPrelievo         := FALSE,
								HmaxElemento			:= WorkAreaState^[Mission^.PPlace].Supporto.HMAX,
								
								Offset_Apprendimento_X 	:= 0,//OffsetApprendimento.Lastra.X, //Offset X Postazione,
								Offset_Apprendimento_Y 	:= TO_REAL(OffsetApprendimento.Lastra.Y), //Offset Y Postazione
								Offset_Apprendimento_Z 	:= TO_REAL(Forming^[WorkAreaState^[Mission^.PPlace].F].PElement[WorkAreaState^[Mission^.PPlace].P].ZDim + OffsetApprendimento.Lastra.Z), //Offset Z Postazione
								Offset_Apprendimento_J 	:= 0,//OffsetApprendimento.Lastra.J, //Offset J Postazione

								Quota_PostX				:= WorkArea^[Mission^.PPlace].X, //Quota X Postazione
								Quota_PostY				:= WorkArea^[Mission^.PPlace].Y, //Quota Y Postazione
								Quota_PostZ				:= WorkArea^[Mission^.PPlace].Z, //Quota Z Postazione
								Quota_PostJ				:= WorkArea^[Mission^.PPlace].Rx, //Quota J Postazione
								
								Offset_Postazione_X 	:= WorkAreaOffset^[Mission^.PPlace].X, //Offset X Postazione
								Offset_Postazione_Y 	:= WorkAreaOffset^[Mission^.PPlace].Y, //Offset Y Postazione
								Offset_Postazione_Z 	:= WorkAreaOffset^[Mission^.PPlace].Z, //Offset Z Postazione
								Offset_Postazione_J 	:= WorkAreaOffset^[Mission^.PPlace].Rx, //Offset J Postazione
								
								Pallet_DimX				:= WorkAreaState^[Mission^.PPlace].Supporto.XDim, //Dimensione X Pallet
								Pallet_DimY				:= WorkAreaState^[Mission^.PPlace].Supporto.YDim, //Dimensione Y Pallet
								Pallet_DimZ				:= WorkAreaState^[Mission^.PPlace].Supporto.ZDim, //Dimensione Z Pallet
								
								Offset_Pallet_X_0		:= 0,//Forming^[WorkAreaState^[Mission^.PPlace].F].Pallet.OFSDE_X0, //Offset X Pallet o Casse
								//Offset_Pallet_Y_0		:= 0,//Forming^[WorkAreaState^[Mission^.PPlace].F].Pallet.OFSDE_Y0, //Offset Y Pallet o Casse 
								//Offset_Pallet_Z_0		:= 0,//Forming^[WorkAreaState^[Mission^.PPlace].F].Pallet.OFSDE_Z0, //Offset Z Pallet o Casse + è grande + il deposito si distanzia dal supporto
								Offset_Pallet_J_0		:= 0,//Forming^[WorkAreaState^[Mission^.PPlace].F].Pallet.OFSDE_J0, //Offset J Pallet o Casse + è grande + la lastra sarà inclinata verso l'angolo crescente
														   
								Offset_Pallet_X_90		:= 0,//Forming^[WorkAreaState^[Mission^.PPlace].F].Pallet.OFSDE_X90, //Offset X Pallet lato 0-90 
								Offset_Pallet_Y_90		:= 0,//Forming^[WorkAreaState^[Mission^.PPlace].F].Pallet.OFSDE_Y90, //Offset Y Pallet lato 0-90 + è grande + il deposito si distanzia dal supporto
								//Offset_Pallet_Z_90		:= 0,//Forming^[WorkAreaState^[Mission^.PPlace].F].Pallet.OFSDE_Z90, //Offset Z Pallet lato 0-90 + è grande + il deposito si distanzia dal supporto
								Offset_Pallet_J_90		:= 0,//Forming^[WorkAreaState^[Mission^.PPlace].F].Pallet.OFSDE_J90, //Offset J Pallet lato 0-90 + è grande + la lastra sarà inclinata in fase di deposito
														  
								Offset_Pallet_X_180		:= 0,//Forming^[WorkAreaState^[Mission^.PPlace].F].Pallet.OFSDE_X180, //Offset X Pallet lato 90-180
								//Offset_Pallet_Y_180		:= OffSetY180Cavallete , //0,//Forming^[WorkAreaState^[Mission^.PPlace].F].Pallet.OFSDE_Y180, //Offset Y Pallet lato 90-180 + è grande + il deposito si distanzia dal supporto
								//Offset_Pallet_Z_180		:= 0,//Forming^[WorkAreaState^[Mission^.PPlace].F].Pallet.OFSDE_Z180, //Offset Z Pallet lato 90-180 + è grande + il deposito si distanzia dal supporto
								Offset_Pallet_J_180		:= 0,//Forming^[WorkAreaState^[Mission^.PPlace].F].Pallet.OFSDE_J180, //Offset J Pallet lato 90-180 + è grande + la lastra sarà inclinata in fase di deposito
								
								Quota_FormaturaX 		:= Forming^[WorkAreaState^[Mission^.PPlace].F].PElement[WorkAreaState^[Mission^.PPlace].P].X, //Quota Deposito X da Formatura
								Quota_FormaturaY 		:= ABS(QuotaLastraYRealTimeDeposito),//ABS(Forming^[WorkAreaState^[Mission^.PPlace].F].PElement[WorkAreaState^[Mission^.PPlace].P].Y), //Quota Deposito Y da Formatura
								Quota_FormaturaZ 		:= ABS(QuotaLastraZRealTimeDeposito),//Forming^[WorkAreaState^[Mission^.PPlace].F].PElement[WorkAreaState^[Mission^.PPlace].P].Z, //Quota Deposito Z da Formatura
								Quota_FormaturaJ 		:= AngoloDepositoLastra,//Forming^[WorkAreaState^[Mission^.PPlace].F].PElement[WorkAreaState^[Mission^.PPlace].P].J, //Quota Deposito Z da Formatura
								
								Distanza_ApproccioFormaturaX 		:= 0,//PickPlaceParameters^.XPlaceApproach,
								Distanza_ApproccioFormaturaY 		:= PickPlaceParameters^.YPlaceApproach, 
								Distanza_ApproccioFormaturaZ 		:= PickPlaceParameters^.ZPlaceApproach,
								Distanza_ApproccioFormaturaJ 		:= 0,//PickPlaceParameters^.JPlaceApproach,

								Quota_DestX 			=> Mission^.XPlace, //Quota DESTINAZIONE X
								Quota_DestY 			=> Mission^.YPlace, //Quota DESTINAZIONE Y
								Quota_DestZ 			=> Mission^.ZPlace, //Quota DESTINAZIONE Z
								Quota_DestJ 			=> Mission^.JPlace, //Quota DESTINAZIONE J	
								
								Quota_ApproccioDestX 	=> Mission^.XPlaceApproach, //Quota APPROCCIO di DESTINAZIONE X
								Quota_ApproccioDestY 	=> Mission^.YPlaceApproach, //Quota APPROCCIO di DESTINAZIONE Y
								Quota_ApproccioDestZ 	=> Mission^.ZPlaceApproach, //Quota APPROCCIO di DESTINAZIONE Z
								Quota_ApproccioDestJ 	=> Mission^.JPlaceApproach);//Quota APPROCCIO di DESTINAZIONE J	

//memorizzo la postazione di deposito
PplaceOld := Mission^.PPlace;
								
IF LatoDeposito = 90 AND WorkAreaState^[Mission^.PPlace].Apprendimento.Z.Lato90.Stato <> APPRENDIMENTO_ESEGUITO THEN
	Mission^.ZPlace := Mission^.ZPlace-50;
END_IF						
															
(* Passo alla pinza i valori di dimensione della lastra *)
ModulePinza^.ElementoInPrelievo.XDim := Mission^.XDim;
ModulePinza^.ElementoInPrelievo.YDim := Mission^.YDim;
ModulePinza^.ElementoInPrelievo.ZDim := Mission^.ZDim;
ModulePinza^.ElementoInPrelievo.Typology := LASTRA;

(* Se il FB di calcolo delle quote Restituisce un errore Mi fermo, altrimenti Eseguo la missione *)
IF TFWAM_CreaMissione_DepLastraDaWA.Errore.Code > 0 THEN
	Errore := TFWAM_CreaMissione_DepLastraDaWA.Errore;
	WorkAreaManager^.State 	:= WAMANAGER_NOP;	// setto lo stato del WAMANAGER
	RestoreCWA^ := TRUE;
	PreviousPWA^ := pwa;
	RETURN;//EXIT;
ELSE
	//IF Mission^.PPick = NumPostazioneDiPareggiatura THEN
	//	WorkAreaManager^.State 	:= WAMANAGER_CICLO_PRELIEVO_LASTRA_DA_PAREGGIATORE_RUN;
	//ELSE
		WorkAreaManager^.State 	:= WAMANAGER_CICLO_PRELIEVO_LASTRA_WA_RUN;
	//END_IF
	RestoreCWA^ := TRUE;
	PreviousPWA^ := pwa;
	RETURN;//EXIT;
END_IF

(* Setto l'uscita che mi determina il deposito del primo pacco in lenta *)
IF WorkAreaState^[Mission^.PPick].Slow = 1 THEN
	DepositoPaccoInLenta := TRUE;
END_IF
END_ACTION

ACTION PREL_DA_PAREGGIATORE_END:
(* Se era settata la velocità lenta di Prelievo pacco, questa viene resettata *)
IF WorkAreaState^[Mission^.PPick].Slow = 1 THEN
	WorkAreaState^[Mission^.PPick].Slow := 0;
	DepositoPaccoInLenta := FALSE;
END_IF
(* Aggiorno la struttura delle Lastre Presenti *)
Mission^.Slab := WorkAreaState^[Mission^.PPick].Slab[NLastraDaPrelevare];
(* Decremento WorkArea^[cwa].P (P=P-1) *)
WorkAreaState^[Mission^.PPick].P := WorkAreaState^[Mission^.PPick].P - 1;

WorkAreaManager^.State 	:= WAMANAGER_CICLO_DEPOSITO_LASTRA_WA_RUN;
RestoreCWA^ := TRUE;
PreviousPWA^ := pwa;
RETURN;//EXIT;
END_ACTION

ACTION PREL_DA_PAREGGIATORE_RUN:
	
IF Mission^.State = MISSION_STATE_PRELIEVO_LASTRA_DA_PAREGGIATORE_RUN THEN
	WorkAreaManager^.State 	:= WAMANAGER_CICLO_PRELIEVO_LASTRA_DA_PAREGGIATORE_RUN;
ELSIF Mission^.State = MISSION_STATE_PRELIEVO_LASTRA_DA_PAREGGIATORE_END THEN
	WorkAreaManager^.State 	:= WAMANAGER_CICLO_PRELIEVO_LASTRA_DA_PAREGGIATORE_END;
ELSIF Mission^.State = MISSION_STATE_ERROR THEN
	;
END_IF
END_ACTION

ACTION PREL_FALDA_END:
CASE TIPO_MAGAZZINO_FALDE OF 
	(* Se il magazzino delle falde è PickPoint *)
	MAGAZZINO_FALDE_IN_PP: 		
		IF WorkPickPoint^[Mission^.PPick].Tipologia = MAGAZZINO_FALDE THEN
			IF WorkPickPoint^[Mission^.PPick].Learned_Z > WorkPickPoint^[Mission^.PPick].Z + Mission^.ZDim THEN
				WorkPickPoint^[Mission^.PPick].Learn_Z 		:= ALTEZZA_CATASTA_FALDE;
				WorkPickPoint^[Mission^.PPick].Learned_Z 	:= ModuleAX_Z^.Ax^.Status.ActPosition; 
				WorkPickPoint^[Mission^.PPick].DoLearn_Z	:= APPRENDIMENTO_ESEGUITO;
			ELSE
				WorkPickPoint^[Mission^.PPick].Learn_Z 		:= ALTEZZA_CATASTA_FALDE;
				WorkPickPoint^[Mission^.PPick].Learned_Z 	:= ALTEZZA_CATASTA_FALDE;
				WorkPickPoint^[Mission^.PPick].DoLearn_Z 	:= APPRENDIMENTO_DA_ESEGUIRE;
				//WorkAreaState^[Mission^.PPick].State := WORKAREA_STATE_OCCUPIED_ENDED;	
			END_IF
		ELSE
			Errore.Code := ErrWAM_PickPoint_NoMagazzinoFalde;//Errore, Il Pick Point, non è di tipo Magazzino Falde
			RETURN;//EXIT;
		END_IF
	(* Se il magazzino delle falde è una WorkArea *)
	MAGAZZINO_FALDE_IN_WA:	
		IF WorkArea^[Mission^.PPick].Typology = TYPOLOGY_LAYER THEN
			IF WorkAreaState^[Mission^.PPick].H > WorkArea^[Mission^.PPick].Z + Mission^.ZDim THEN
				WorkAreaState^[Mission^.PPick].H 			:= ModuleAX_Z^.Ax^.Status.ActPosition; 
				WorkAreaState^[Mission^.PPick].Apprendimento.Z.Lato0.QuotaStart 	:= ALTEZZA_CATASTA_FALDE;
				WorkAreaState^[Mission^.PPick].Apprendimento.Z.Lato0.QuotaRilevata 	:= ModuleAX_Z^.Ax^.Status.ActPosition;
				WorkAreaState^[Mission^.PPick].Apprendimento.Z.Lato0.Stato		 	:= APPRENDIMENTO_ESEGUITO;
			ELSE
				WorkAreaState^[Mission^.PPick].H 			:= WorkArea^[Mission^.PPick].Z;
				WorkAreaState^[Mission^.PPick].Apprendimento.Z.Lato0.QuotaStart 	:= ALTEZZA_CATASTA_FALDE;
				WorkAreaState^[Mission^.PPick].Apprendimento.Z.Lato0.QuotaRilevata 	:= ALTEZZA_CATASTA_FALDE;
				WorkAreaState^[Mission^.PPick].Apprendimento.Z.Lato0.Stato		 	:= APPRENDIMENTO_DA_ESEGUIRE;
				//WorkAreaState^[Mission^.PPick].State := WORKAREA_STATE_OCCUPIED_ENDED;	
			END_IF
			(* Aggiorno la struttura delle Lastre Presenti *)
			Mission^.Slab := WorkAreaState^[Mission^.PPick].Slab[NLastraDaPrelevare];
			(* Decremento WorkArea^[cwa].P (P=P-1) *)
			WorkAreaState^[Mission^.PPick].P := WorkAreaState^[Mission^.PPick].P - 1;
		ELSE
			Errore.Code := ErrWAM_WorkArea_NoMagazzinoFalde; // Errore, la WorkArea non è di tipo Magazzino Falde
			RETURN;//	EXIT;
		END_IF
ELSE
	Errore.Code := ErrWAM_TipologiaMagazzinoFaldaNONRiconosciuta;// Errore, Nell'impianto è stata impostata una tipologia di magazzino falde non prevista!!!
	RETURN;//EXIT;		
END_CASE
WorkAreaManager^.State 	:= WAMANAGER_CICLO_DEPOSITO_FALDA_RUN;
RestoreCWA^ := TRUE;
PreviousPWA^ := pwa;
RETURN;//EXIT;
END_ACTION

ACTION PREL_FALDA_RUN:
IF Mission^.State = MISSION_STATE_PRELIEVO_FALDA_RUN THEN
	WorkAreaManager^.State := WAMANAGER_CICLO_PRELIEVO_FALDA_RUN;
ELSIF Mission^.State = MISSION_STATE_PRELIEVO_FALDA_END THEN
	WorkAreaManager^.State := WAMANAGER_CICLO_PRELIEVO_FALDA_END;
	RestoreCWA^ := TRUE;
	PreviousPWA^ := pwa;
	RETURN;//EXIT;
ELSIF Mission^.State = MISSION_STATE_ERROR THEN
	;
END_IF
END_ACTION

ACTION PREL_LASTRA_PP_END:
(* Se era settata la velocità lenta di Prelievo pacco, questa viene resettata *)
IF WorkAreaState^[Mission^.PPick].Slow = 1 THEN
	WorkAreaState^[Mission^.PPick].Slow := 0;
	DepositoPaccoInLenta := FALSE;
END_IF

(* Aggiorno Altezza Pallet su Ultima Lastra depositata *)
(*!!!!!!!!!!! ATTUALMENTE CI BASIAMO SULLE QUOTE INVIATE DA HMI PER IL DEPOSITO E ANDIAMO IN TASTEGGIO, LE CASSE SONO PIU' ALTE DELLA LASTRA DEPOSITATA E 
IN CASO DI CAVALLETTO L'ALTEZZA E' FISSA... QUINDI, NON AGGIORNIAMO NESSUNA ALTEZZA!!!!!*)
(**IF AbilitaAggiornamento_AltezzaWA_ConQuotaAsseZ THEN
	WorkArea^[Mission^.PPlace].H := ModuloAsse_Z.Ax^.Status.ActPosition;
ELSE
	WorkArea^[Mission^.PPlace].H := WorkArea^[Mission^.PPlace].HPL + 
									Forming^[WorkAreaState^[Mission^.PPlace].F].PackXP[WorkAreaState^[Mission^.PPlace].P].Z;
END_IF**)			
CASE TIPOLOGIA_FUNZIONAMENTO_MACCHINA OF
	FUNZIONAMENTO_PALLETTIZZATORE:
									WorkAreaManager^.State 	:= WAMANAGER_CICLO_DEPOSITO_LASTRA_PP_RUN;
									RestoreCWA^ 	:= TRUE;
									PreviousPWA^ 	:= pwa;
									RETURN;//EXIT;
							
ELSE
	CASE WorkAreaProductionList^[cwa].PElementList[WorkAreaState^[Mission^.PPlace].P].Pareggiatura OF
		(* Se la Pareggiatura della Lastra è Disabilitata *)
		PAREGGIATURA_DISABILITATA:
									WorkAreaManager^.State 	:= WAMANAGER_CICLO_DEPOSITO_LASTRA_PP_RUN;
									RestoreCWA^ := TRUE;
									PreviousPWA^ := pwa;
									RETURN;//EXIT;
									
		(* Se la Pareggiatura della Lastra è Abilitata e da Eseguire *)
		PAREGGIATURA_DA_ESEGUIRE:
									Mission^.PPlace := NumPostazioneDiPareggiatura;
									(* Valorizzazione quote di deposito Ciclo Lastra *)
									TFWAM_CreaMissione_DepLastraDaWA(NPosInLavoro			:= Mission^.PPlace, //Numero Postazione di depositio
																		Angolo_Destinazione 		:= Forming^[WorkAreaState^[Mission^.PPlace].F].PElement[WorkAreaState^[Mission^.PPlace].P].J, //Angolo di deposito dell'elemento
																		PosizioneAttuale_X      := ModuleAX_X^.Ax^.Status.ActPosition, //Posizione attuale asse X
																		TipologiaTraiettoria    := Forming^[WorkAreaState^[cwa].F].PElement[WorkAreaState^[cwa].P].Trajectory,
																			
																		Quota_PostX				:= WorkArea^[Mission^.PPlace].X, //Quota X Postazione
																		Quota_PostY				:= WorkArea^[Mission^.PPlace].Y, //Quota Y Postazione
																		Quota_PostZ				:= WorkArea^[Mission^.PPlace].Z, //Quota Z Postazione
																		Quota_PostJ				:= WorkArea^[Mission^.PPlace].Rx, //Quota J Postazione
																		
																		Offset_Postazione_X 	:= WorkAreaOffset^[Mission^.PPlace].X, //Offset X Postazione
																		Offset_Postazione_Y 	:= WorkAreaOffset^[Mission^.PPlace].Y, //Offset Y Postazione
																		Offset_Postazione_Z 	:= WorkAreaOffset^[Mission^.PPlace].Z, //Offset Z Postazione
																		Offset_Postazione_J 	:= WorkAreaOffset^[Mission^.PPlace].Rx, //Offset J Postazione
																		
																		Pallet_DimX				:= Forming^[WorkAreaState^[Mission^.PPlace].F].Pallet.XDim, //Dimensione X Pallet
																		Pallet_DimY				:= Forming^[WorkAreaState^[Mission^.PPlace].F].Pallet.YDim, //Dimensione Y Pallet
																		Pallet_DimZ				:= Forming^[WorkAreaState^[Mission^.PPlace].F].Pallet.ZDim, //Dimensione Z Pallet
																		
																		Offset_Pallet_X_0		:= Forming^[WorkAreaState^[Mission^.PPlace].F].Pallet.OFSDE_X0, //Offset X Pallet o Casse
																		Offset_Pallet_Y_0		:= Forming^[WorkAreaState^[Mission^.PPlace].F].Pallet.OFSDE_Y0, //Offset Y Pallet o Casse 
																		Offset_Pallet_Z_0		:= Forming^[WorkAreaState^[Mission^.PPlace].F].Pallet.OFSDE_Z0, //Offset Z Pallet o Casse + è grande + il deposito si distanzia dal supporto
																		Offset_Pallet_J_0		:= Forming^[WorkAreaState^[Mission^.PPlace].F].Pallet.OFSDE_J0, //Offset J Pallet o Casse + è grande + la lastra sarà inclinata verso l'angolo crescente
																		
																		Offset_Pallet_X_90		:= Forming^[WorkAreaState^[Mission^.PPlace].F].Pallet.OFSDE_X90, //Offset X Pallet lato 0-90 
																		Offset_Pallet_Y_90		:= Forming^[WorkAreaState^[Mission^.PPlace].F].Pallet.OFSDE_Y90, //Offset Y Pallet lato 0-90 + è grande + il deposito si distanzia dal supporto
																		Offset_Pallet_Z_90		:= Forming^[WorkAreaState^[Mission^.PPlace].F].Pallet.OFSDE_Z90, //Offset Z Pallet lato 0-90 + è grande + il deposito si distanzia dal supporto
																		Offset_Pallet_J_90		:= Forming^[WorkAreaState^[Mission^.PPlace].F].Pallet.OFSDE_J90, //Offset J Pallet lato 0-90 + è grande + la lastra sarà inclinata in fase di deposito
																		
																		Offset_Pallet_X_180		:= Forming^[WorkAreaState^[Mission^.PPlace].F].Pallet.OFSDE_X180, //Offset X Pallet lato 90-180
																		Offset_Pallet_Y_180		:= Forming^[WorkAreaState^[Mission^.PPlace].F].Pallet.OFSDE_Y180, //Offset Y Pallet lato 90-180 + è grande + il deposito si distanzia dal supporto
																		Offset_Pallet_Z_180		:= Forming^[WorkAreaState^[Mission^.PPlace].F].Pallet.OFSDE_Z180, //Offset Z Pallet lato 90-180 + è grande + il deposito si distanzia dal supporto
																		Offset_Pallet_J_180		:= Forming^[WorkAreaState^[Mission^.PPlace].F].Pallet.OFSDE_J180, //Offset J Pallet lato 90-180 + è grande + la lastra sarà inclinata in fase di deposito
																		
																		Quota_FormaturaX 		:= Forming^[WorkAreaState^[Mission^.PPlace].F].PElement[WorkAreaState^[Mission^.PPlace].P].X, //Quota Deposito X da Formatura
																		Quota_FormaturaY 		:= Forming^[WorkAreaState^[Mission^.PPlace].F].PElement[WorkAreaState^[Mission^.PPlace].P].Y, //Quota Deposito Y da Formatura
																		Quota_FormaturaZ 		:= Forming^[WorkAreaState^[Mission^.PPlace].F].PElement[WorkAreaState^[Mission^.PPlace].P].Z, //Quota Deposito Z da Formatura
																		Quota_FormaturaJ 		:= Forming^[WorkAreaState^[Mission^.PPlace].F].PElement[WorkAreaState^[Mission^.PPlace].P].J, //Quota Deposito Z da Formatura
																		
																		Distanza_ApproccioFormaturaX 		:= Forming^[WorkAreaState^[Mission^.PPlace].F].PElement[WorkAreaState^[Mission^.PPlace].P].AX, //Quota Deposito X da Formatura
																		Distanza_ApproccioFormaturaY 		:= Forming^[WorkAreaState^[Mission^.PPlace].F].PElement[WorkAreaState^[Mission^.PPlace].P].AY, //Quota Deposito Y da Formatura
																		Distanza_ApproccioFormaturaZ 		:= Forming^[WorkAreaState^[Mission^.PPlace].F].PElement[WorkAreaState^[Mission^.PPlace].P].AZ, //Quota Deposito Z da Formatura
																		Distanza_ApproccioFormaturaJ 		:= Forming^[WorkAreaState^[Mission^.PPlace].F].PElement[WorkAreaState^[Mission^.PPlace].P].AJ, //Quota Deposito Z da Formatura
																		
																		Quota_DestX 			=> Mission^.XPlace, //Quota DESTINAZIONE X
																		Quota_DestY 			=> Mission^.YPlace, //Quota DESTINAZIONE Y
																		Quota_DestZ 			=> Mission^.ZPlace, //Quota DESTINAZIONE Z
																		Quota_DestJ 			=> Mission^.JPlace, //Quota DESTINAZIONE J	
																		
																		Quota_ApproccioDestX 	=> Mission^.XPlaceApproach, //Quota APPROCCIO di DESTINAZIONE X
																		Quota_ApproccioDestY 	=> Mission^.YPlaceApproach, //Quota APPROCCIO di DESTINAZIONE Y
																		Quota_ApproccioDestZ 	=> Mission^.ZPlaceApproach, //Quota APPROCCIO di DESTINAZIONE Z
																		Quota_ApproccioDestJ 	=> Mission^.JPlaceApproach);//Quota APPROCCIO di DESTINAZIONE J		
			IF TFWAM_CreaMissione_DepLastraDaWA.Errore.Code > 0 THEN
				WorkAreaManager^.State 	:= WAMANAGER_NOP;	// setto lo stato del WAMANAGER
				RETURN;//EXIT;
			ELSE
				WorkAreaManager^.State 	:= WAMANAGER_CICLO_DEPOSITO_LASTRA_SU_PAREGGIATORE_RUN;
				RestoreCWA^ := TRUE;
				PreviousPWA^ := pwa;
				RETURN;//EXIT;
			END_IF	
	ELSE
		;
	END_CASE
END_CASE
END_ACTION

ACTION PREL_LASTRA_PP_RUN:

IF Mission^.State = MISSION_STATE_PRELIEVO_LASTRA_PP_RUN THEN
	;
ELSIF Mission^.State = MISSION_STATE_PRELIEVO_LASTRA_PP_END THEN
	WorkAreaManager^.State 	:= WAMANAGER_CICLO_PRELIEVO_LASTRA_PP_END;
ELSIF Mission^.State = MISSION_STATE_ERROR THEN
	;
END_IF
END_ACTION

ACTION PREL_LASTRA_WA_END:

(* Imposto lo stato dell' apprendimento *)
CASE LatoPrelievo OF			
	0:
		IF WorkAreaState^[Mission^.PPICk].Apprendimento.Y.Lato0.Stato <> APPRENDIMENTO_ESEGUITO THEN
			WorkAreaState^[Mission^.PPICk].Apprendimento.Y.Lato0.Stato := APPRENDIMENTO_ESEGUITO;
			WorkAreaState^[Mission^.PPICk].Apprendimento.Y.Lato0.QuotaRilevata := ModuleAX_Y^.QuotaAsseLetturaTasteggio;
		ELSE
			WorkAreaState^[Mission^.PPICk].Apprendimento.Y.Lato0.QuotaRilevata := ModuleAX_Y^.QuotaAsseLetturaTasteggio;
		END_IF
		
	90:
		IF  WorkAreaState^[Mission^.PPICk].Apprendimento.Z.Lato90.Stato <> APPRENDIMENTO_ESEGUITO THEN
			WorkAreaState^[Mission^.PPICk].Apprendimento.Z.Lato90.Stato 				:= APPRENDIMENTO_ESEGUITO;
			WorkAreaState^[Mission^.PPICk].Apprendimento.Z.Lato90.QuotaRilevata 		:= ModuleAX_Z^.QuotaAsseLetturaTasteggio;
			WorkAreaState^[Mission^.PPICk].Supporto.HMAX 	:=  MAX(WorkAreaState^[Mission^.PPick].Supporto.HMAX,ModuleAX_Z^.QuotaAsseLetturaTasteggio);
			WorkAreaState^[Mission^.PPICk].H 				:=  ModuleAX_Z^.QuotaAsseLetturaTasteggio;
			WorkAreaState^[Mission^.PPICk].HPL 				:=  ModuleAX_Z^.QuotaAsseLetturaTasteggio;	 

		ELSE
			WorkAreaState^[Mission^.PPick].Apprendimento.Z.Lato90.Stato 				:= 	APPRENDIMENTO_ESEGUITO;
			WorkAreaState^[Mission^.PPick].Apprendimento.Z.Lato90.QuotaRilevata 		:=  ModuleAX_Z^.QuotaAsseLetturaTasteggio;
			WorkAreaState^[Mission^.PPick].Supporto.HMAX 	:=  MAX(WorkAreaState^[Mission^.PPick].Supporto.HMAX,ModuleAX_Z^.QuotaAsseLetturaTasteggio);
			WorkAreaState^[Mission^.PPick].H 				:=  ModuleAX_Z^.QuotaAsseLetturaTasteggio;
			WorkAreaState^[Mission^.PPick].HPL 				:=  ModuleAX_Z^.QuotaAsseLetturaTasteggio;	 

		END_IF
		
	180:
		IF WorkAreaState^[Mission^.PPick].Apprendimento.Y.Lato180.Stato <> APPRENDIMENTO_ESEGUITO THEN
			WorkAreaState^[Mission^.PPick].Apprendimento.Y.Lato180.Stato := APPRENDIMENTO_ESEGUITO;
			WorkAreaState^[Mission^.PPick].Apprendimento.Y.Lato180.QuotaRilevata := ModuleAX_Y^.QuotaAsseLetturaTasteggio;
		ELSE
			WorkAreaState^[Mission^.PPick].Apprendimento.Y.Lato180.QuotaRilevata := ModuleAX_Y^.QuotaAsseLetturaTasteggio;
		END_IF
END_CASE

(* Se era settata la velocità lenta di Prelievo pacco, questa viene resettata *)
IF WorkAreaState^[Mission^.PPick].Slow = 1 THEN
	WorkAreaState^[Mission^.PPick].Slow := 0;
	DepositoPaccoInLenta := FALSE;
END_IF

(* Aggiorno Altezza Pallet su Ultima Lastra depositata *)
(*!!!!!!!!!!! ATTUALMENTE CI BASIAMO SULLE QUOTE INVIATE DA HMI PER IL DEPOSITO E ANDIAMO IN TASTEGGIO, LE CASSE SONO PIU' ALTE DELLA LASTRA DEPOSITATA E 
IN CASO DI CAVALLETTO L'ALTEZZA E' FISSA... QUINDI, NON AGGIORNIAMO NESSUNA ALTEZZA!!!!!*)
(**IF AbilitaAggiornamento_AltezzaWA_ConQuotaAsseZ THEN
	WorkArea^[Mission^.PPlace].H := ModuloAsse_Z.Ax^.Status.ActPosition;
ELSE
	WorkArea^[Mission^.PPlace].H := WorkArea^[Mission^.PPlace].HPL + 
									Forming^[WorkAreaState^[Mission^.PPlace].F].PackXP[WorkAreaState^[Mission^.PPlace].P].Z;
END_IF**)


WorkAreaState^[Mission^.PPick].P := WorkAreaState^[Mission^.PPick].P - 1;
IF WorkAreaState^[Mission^.PPick].Supporto.Tipologia = CAVALLETTO THEN 
	IF PosicionJOrigen = 0 THEN 
		WorkAreaState^[Mission^.PPick].P_Cava.HMI_NumeroPezziPresentiPostazione_A_Cavaleto := WorkAreaState^[Mission^.PPick].P_Cava.HMI_NumeroPezziPresentiPostazione_A_Cavaleto -1 ;
	ELSIF PosicionJOrigen = 180 THEN 	
		WorkAreaState^[Mission^.PPick].P_Cava.HMI_NumeroPezziPresentiPostazione_B_Cavaleto := WorkAreaState^[Mission^.PPick].P_Cava.HMI_NumeroPezziPresentiPostazione_B_Cavaleto -1 ;
	END_IF
END_IF

WorkAreaManager^.State 	:= WAMANAGER_CICLO_DEPOSITO_LASTRA_WA_RUN;
RestoreCWA^ := TRUE;
PreviousPWA^ := pwa;
RETURN;//EXIT;
END_ACTION

ACTION PREL_LASTRA_WA_RUN:
IF Mission^.State = MISSION_STATE_PRELIEVO_LASTRA_WA_RUN THEN
	;
ELSIF Mission^.State = MISSION_STATE_PRELIEVO_LASTRA_WA_END THEN
	WorkAreaManager^.State 	:= WAMANAGER_CICLO_PRELIEVO_LASTRA_WA_END;
ELSIF Mission^.State = MISSION_STATE_ERROR THEN
	;
END_IF
END_ACTION

END_FUNCTION_BLOCK

(* stored: Version 1.1.0.1, ProductVersion 3.1.4024.11
   POU TFPalletizerWorkAreaManagerTF_Lastre: Id {02c9f462-c94d-4b6f-b759-73bc34ee33fa}, SpecialFunc None
   Folder FALDA: Id {ae00f510-4b52-40ac-b057-b96211686c69}
   Folder LASTRA: Id {243b257f-fd69-499e-8317-24f5934ef8fe}
   Folder Pareggiatore: Id {d964441b-bb28-4fba-b1f2-33523b9e15a1}
   Folder PickPoint: Id {ba29b62a-01f3-48a1-8aa2-964bb0a791d6}
   Folder WorkArea: Id {2ef04b7d-b074-4c1d-945d-cab697d34ea3}
   Folder PAREGGIATORE: Id {901eb3b9-3249-43d7-a039-22fc0b813877}
   Folder RIPOSO: Id {e0368fa6-8cdf-4171-80ea-8a3358a01de2}
   Action CICLO_PAREGGIATURA_END: Id {ea110164-1c85-4d1c-bd0c-a01ccaa803d8}
   Action CICLO_PAREGGIATURA_RUN: Id {48209740-0a10-4b1c-b0a8-4cc33eab97f2}
   Action DEP_FALDA_END: Id {d3a53a5f-9ff5-4df9-9ae3-4dc6654a3c65}
   Action DEP_FALDA_RUN: Id {f903c77b-e098-43cf-8c7d-5c88a0586800}
   Action DEP_LASTRA_PP_END: Id {692279df-5b0f-48e2-8e6f-abdf1b00835b}
   Action DEP_LASTRA_PP_RUN: Id {30acaa4c-a2ed-4beb-ae76-26b76d953a2a}
   Action DEP_LASTRA_WA_END: Id {587a21ea-99be-424c-bf07-0061766337df}
   Action DEP_LASTRA_WA_RUN: Id {df76aedf-577c-4d47-bed3-bf49ba2e3d75}
   Action DEP_PAREGGIATORE_RUN: Id {067c5f0a-10d6-4320-9740-23482174cf77}
   Action DEP_SU_PAREGGIATORE_END: Id {1c09f636-e5de-4f0e-bbac-d10d3262ffec}
   Action DEP_SU_PAREGGIATORE_RUN: Id {721797e8-74d3-45b0-b6d4-6a337ea45850}
   Action FALDA_INIT: Id {5762d4e9-6314-4eb3-b497-1fb6ed1926c5}
   Action LASTRA_PP_INIT: Id {8c3ab7d6-65f9-452d-a9ea-353a875d31e9}
   Action LASTRA_WA_INIT: Id {972dc595-b257-4443-ad76-c610d7b6e262}
   Action PREL_DA_PAREGGIATORE_END: Id {95350da3-6268-40e4-82d6-8c1d7fa2d160}
   Action PREL_DA_PAREGGIATORE_RUN: Id {df32ea60-f9f5-4b2e-acfc-28a07e09c64d}
   Action PREL_FALDA_END: Id {432b773c-53d0-4572-8773-28b2a1cbd6b4}
   Action PREL_FALDA_RUN: Id {a30b094f-e701-4e4e-b5e6-b4731ca76176}
   Action PREL_LASTRA_PP_END: Id {e1b25cfa-705a-402a-99f7-1ad057e3d370}
   Action PREL_LASTRA_PP_RUN: Id {194006f4-1041-48b1-b841-6e21804fd0bf}
   Action PREL_LASTRA_WA_END: Id {83317d89-60dd-48a2-a005-0e5a1034f3dd}
   Action PREL_LASTRA_WA_RUN: Id {77e8b8aa-1944-4bc5-9ce7-7ff8cc835ab8} *)
